// TIA Portal V17 export
// export: Created 2023-08-28T08:18:09.2848054Z, ExportSetting WithDefaults, DisplayName Totally Integrated Automation Portal, DisplayVersion V17 Update 5, DisplayName TIA Portal Openness, DisplayVersion V17 Update 5, DisplayName TIA Portal Teamcenter Gateway, DisplayVersion V17 Update 5, DisplayName TIA Portal Version Control Interface, DisplayVersion V17, DisplayName Simotion SCOUT TIA, DisplayVersion 5.4.3.0, DisplayName TIA Portal Test Suite Advanced, DisplayVersion V17 Update 1, DisplayName SIMOCODE ES, DisplayVersion V17 Update 5, DisplayName SINAMICS Startdrive Advanced, DisplayVersion V17 SP1, DisplayName SINAMICS Startdrive G130, G150, S120, S150, SINAMICS MV, S210, DisplayVersion V17 SP1, DisplayName SINAMICS Startdrive G110M, G120, G120C, G120D, G120P, G115D, DisplayVersion V17 SP1, DisplayName SIRIUS Safety ES, DisplayVersion V17 Update 5, DisplayName STEP 7 Professional, DisplayVersion V17 Update 5, DisplayName STEP 7 CFC, DisplayVersion V17 Update 1, DisplayName STEP 7 Safety, DisplayVersion V17, DisplayName WinCC Advanced, DisplayVersion V17 Update 5, DisplayName SIMATIC Visualization Architect, DisplayVersion V17 Update 5
FUNCTION "05_Output Feedback" : Void   // FC6, F_FBD
TITLE = Manage Safety Outputs
{ S7_Optimized_Access := 'TRUE' }
VERSION : 0.1
// stored: AutoNumber true, IsIECCheckEnabled false, UDAEnableTagReadback false
   VAR_TEMP
      DU_EX : Bool;
      ISPC_EX : Bool;
      ZONE_EX : Bool;
   END_VAR
BEGIN

REGION Network 1: !!COLUMN_1!!
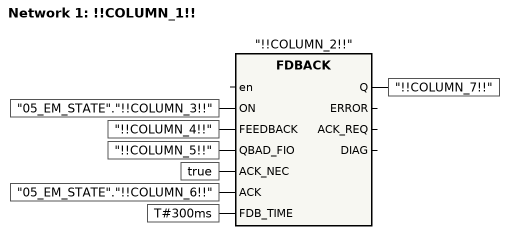
   "!!COLUMN_2!!"(ON := "05_EM_STATE"."!!COLUMN_3!!",   // FDBACK
                  FEEDBACK := "!!COLUMN_4!!",
                  QBAD_FIO := "!!COLUMN_5!!",
                  ACK_NEC := true,
                  ACK := "05_EM_STATE"."!!COLUMN_6!!",
                  FDB_TIME := T#300ms,
                  Q => "!!COLUMN_7!!");
END_REGION
END_FUNCTION
